TYPE stMotor :	
STRUCT
	Name				: STRING;
	TestModeActive		: BOOL;
	UseReverse			: BOOL;
	iTestForward		: BOOL;
	iTestReverse		: BOOL;
	oMoveForward		: BOOL;
	oMoveReverse		: BOOL;
	oResetError			: BOOL;
	Status_MotorRunning	: BOOL;
	Status_Error		: BOOL;
	ErrorID				: UINT;
END_STRUCT
END_TYPE

(* stored: Version 1.1.0.1, ProductVersion 3.1.4024.9
   DUT stMotor: Id {ef5af004-a7f1-4fad-baa0-4649d059c060} *)
